{attribute addProperty BoxType "IODEVICETYPE_ETHERCATPROT"}
{attribute addProperty Id "TcTerminals210_1EK1100TcTerminals210_1EK1100_99191ECD00SyncUnitsSyncUnits_3FA29F3C21627InputsInputs_C75D3FEC1280160OutputsOutputs_47D1E803848106InfoDataInfoData_45F98C5022428"}
{attribute addProperty CRC "246358054"}
{attribute addProperty SizeInBites "2568"}
{attribute addProperty SizeInBytes "321"}
TYPE EtherCAT_Master_KLxxxx_1_0EAF2026 :
STRUCT
	{attribute addProperty Name "TcTerminals210_1EK1100"}
	TcTerminals210_1EK1100 : TcTerminals210_1EK1100_99191ECD;
	{attribute addProperty Name "SyncUnits"}
	SyncUnits : SyncUnits_3FA29F3C;
	{attribute addProperty Name "Inputs"}
	Inputs : Inputs_C75D3FEC;
	{attribute addProperty Name "Outputs"}
	Outputs : Outputs_47D1E803;
	{attribute addProperty Name "InfoData"}
	InfoData : InfoData_45F98C50;
END_STRUCT
END_TYPE

(* stored: Version 1.2.0.0, ProductVersion 3.1.4024.9
   DUT EtherCAT_Master_KLxxxx_1_0EAF2026: Id {b5a00e5a-25d4-43e1-b817-f6668342c3b4} *)
